PROGRAM P_DimmingLight_Test_ST
VAR
	fbDimmingLight		:	FB_DimmingLight;
	bOn					:	BOOL;
	bOff				:	BOOL;
	bRecallMinLevel		:	BOOL;
	bSetControlLevel	:	BOOL;
	nSetControlLevel	:	BYTE;
	bControlLevel		:	BOOL;
	nControlLevel		:	BYTE;
END_VAR

fbDimmingLight();

IF (bOn) THEN
	fbDimmingLight.M_On();
	bOn := FALSE;
END_IF
IF (bOff) THEN
	fbDimmingLight.M_Off();
	bOff := FALSE;
END_IF
IF (bRecallMinLevel) THEN
	fbDimmingLight.M_RecallMinLevel();
	bRecallMinLevel := FALSE;
END_IF
IF (bSetControlLevel) THEN
	fbDimmingLight.M_SetControlLevel(nSetControlLevel);
	bSetControlLevel := FALSE;
END_IF

bControlLevel := fbDimmingLight.bControlLevel;
nControlLevel := fbDimmingLight.nControlLevel;

END_PROGRAM

(* stored: Version 1.1.0.1, ProductVersion 3.1.0.23
   POU P_DimmingLight_Test_ST: Id {a0f539b5-31a1-424d-9748-dd8f15a48a5e} *)
